# EPICS substitutions: iocBoot/iocLakeShore/lakeshore.substitutions
file "${TOP}/db/lakeshore336.template"
{
pattern {   P,      PORT,   ADDR, TEMPSCAN, SCAN}
	    {"COMP:A", "L0",    "0",   "1",    "5" }
}

file "${TOP}/db/lakeshore336output.template"
{
pattern {   P,       OUT,   PORT,   ADDR, TEMPSCAN, SCAN}
	    {"COMP:A",   "1",   "L0",    "0",   "1",    "5" }
}

#file "${TOP}/db/save_restoreStatus.db"
#{
#pattern {    P    }
#        {"COMP:A:"}
#}
